TYPE "EFC_EX_STATUS_WORD"
VERSION : 0.1
// Block: EFC_EX_STATUS_WORD
   STRUCT
      Reserved0 : Bool;
      Reserved1 : Bool;
      Reserved2 : Bool;
      Reserved3 : Bool;
      Reserved4 : Bool;
      Reserved5 : Bool;
      Warning : Bool;
      Reserved7 : Bool;
      Mode24V : Bool;
      SleepMode : Bool;
      ConverterOk : Bool;
      Reserved11 : Bool;
      Reserved12 : Bool;
      Reserved13 : Bool;
      Reserved14 : Bool;
      Reserved15 : Bool;
   END_STRUCT;

END_TYPE
